{attribute 'enable_dynamic_creation'}
FUNCTION_BLOCK FB_TargetManager
VAR
	// TODO: Replace with proper array size or dynamic list
	_targets : ARRAY[1..100] OF ST_Target;
	_targetCount : INT := 0;
END_VAR

// TargetManager implementation

METHOD PUBLIC AddTarget : BOOL
VAR_INPUT
	target : ST_Target;
END_VAR
IF _targetCount < 100 THEN
	_targetCount := _targetCount + 1;
	_targets[_targetCount] := target;
	AddTarget := TRUE;
ELSE
	AddTarget := FALSE;
END_IF
END_METHOD

METHOD PUBLIC RemoveTarget : BOOL
VAR_INPUT
	target : ST_Target;
END_VAR
VAR
	i : INT;
END_VAR
// TODO: Implement target removal
RemoveTarget := FALSE;
END_METHOD

METHOD PUBLIC UpdateTarget : BOOL
VAR_INPUT
	target : ST_Target;
END_VAR
// TODO: Implement target update
UpdateTarget := FALSE;
END_METHOD

METHOD PUBLIC GetTargetByName : BOOL
VAR_INPUT
	sName : STRING(80);
END_VAR
VAR_OUTPUT
	target : ST_Target;
END_VAR
VAR
	i : INT;
END_VAR
FOR i := 1 TO _targetCount DO
	IF _targets[i].name = sName THEN
		target := _targets[i];
		GetTargetByName := TRUE;
		RETURN;
	END_IF
END_FOR
GetTargetByName := FALSE;
END_METHOD

METHOD PUBLIC GetAllTargets : INT
VAR_OUTPUT
	// TODO: Use proper return type (List<Target> not supported in IEC 61131-3)
	// For now returning count
END_VAR
GetAllTargets := _targetCount;
END_METHOD

END_FUNCTION_BLOCK

(* stored: Version 1.1.0.1
   POU FB_TargetManager: Id {e1b2c3d4-2222-2222-2222-222222222222}
   Method AddTarget: Id {e1b2c3d4-2221-2222-2222-222222222222}
   Method RemoveTarget: Id {e1b2c3d4-2222-2222-2222-222222222222}
   Method UpdateTarget: Id {e1b2c3d4-2223-2222-2222-222222222222}
   Method GetTargetByName: Id {e1b2c3d4-2224-2222-2222-222222222222}
   Method GetAllTargets: Id {e1b2c3d4-2225-2222-2222-222222222222} *)
